(* PLC project DisabledLabelFixture, CODESYS CODESYS V3.5 SP11 *)
(* stored: creationDateTime 2026-09-12T00:00:00 *)

PROGRAM DISABLED_LABEL
  VAR
    xA : BOOL;
    oA : BOOL;
    xB : BOOL;
    oB : BOOL;
  END_VAR

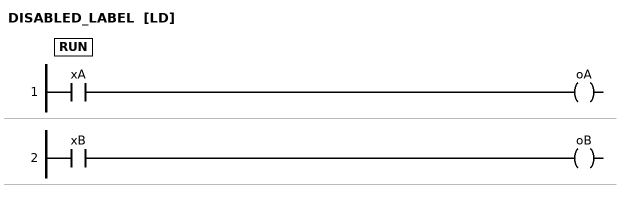
(* LD diagram, written out as Structured Text *)

RUN:
oA := xA;

oB := xB;
END_PROGRAM
